INTERFACE ITF_ErrorHandlerSubject

METHOD AttachDevice : BOOL
VAR_INPUT
	itfDevice 	: ITF_Device;
END_VAR
END_METHOD

END_INTERFACE

(* stored: Version 1.1.0.1, ProductVersion 3.1.4024.11
   Itf ITF_ErrorHandlerSubject: Id {e353ff13-2755-43fd-b4d5-b805969a0255}
   Method AttachDevice: Id {08238ad0-a076-4f1b-ae95-df11cc8dfb7d} *)
